# EPICS substitutions: ek9000App/Db/EL1712.substitutions
file EL1712.template
{ 	pattern
	{
		TERMINAL,

	}
	{
	}
}
